(* PLC project Blank Project, Blank Blank 1.0 *)
(* stored: creationDateTime 2016-05-18T21:14:07, modificationDateTime 2020-07-06T15:08:10 *)

PROGRAM My_Program
  VAR
    flow_in AT %IW0 : INT;
    flow_out AT %IW1 : INT;
    ug_opcmd AT %QX0.0 : BOOL;
    ug_clcmd AT %QX0.1 : BOOL;
    ug_val AT %IW2 : INT;
    lg_opcmd AT %QX0.2 : BOOL;
    lg_clcmd AT %QX0.3 : BOOL;
    lg_val AT %IW3 : INT;
    uv_opcmd AT %QX0.4 : BOOL;
    uv_clcmd AT %QX0.5 : BOOL;
    uv_val AT %IW4 : INT;
    lv_opcmd AT %QX0.6 : BOOL;
    lv_clcmd AT %QX0.7 : BOOL;
    lv_val AT %IW5 : INT;
    dp_chmbr AT %IW6 : INT;
    dp_rsvr AT %IW7 : INT := 4200;
    dp_tlwtr AT %IW8 : INT;
    warn_btn AT %QX1.0 : BOOL;
    em_gt AT %QX1.1 : BOOL;
    em_vlv AT %QX1.2 : BOOL;
    ht_still AT %IW9 : INT := 2150;
    dprel_rsvr AT %QW0 : INT;
    rsrvr_eq AT %QX1.3 : BOOL;
    tlwtr_eq AT %QX1.4 : BOOL;
  END_VAR
  VAR
    TP0 : TP;
    TP1 : TP;
    TP2 : TP;
  END_VAR
  VAR  (* added by the conversion: wires and edge detectors of the diagram *)
    _XOR35_OUT : BOOL;
    _DIV140_OUT : REAL;
    _XOR28_OUT : BOOL;
    _DIV17_OUT : REAL;
    _XOR57_OUT : BOOL;
    _DIV144_OUT : REAL;
    _XOR83_OUT : BOOL;
    _DIV79_OUT : REAL;
  END_VAR

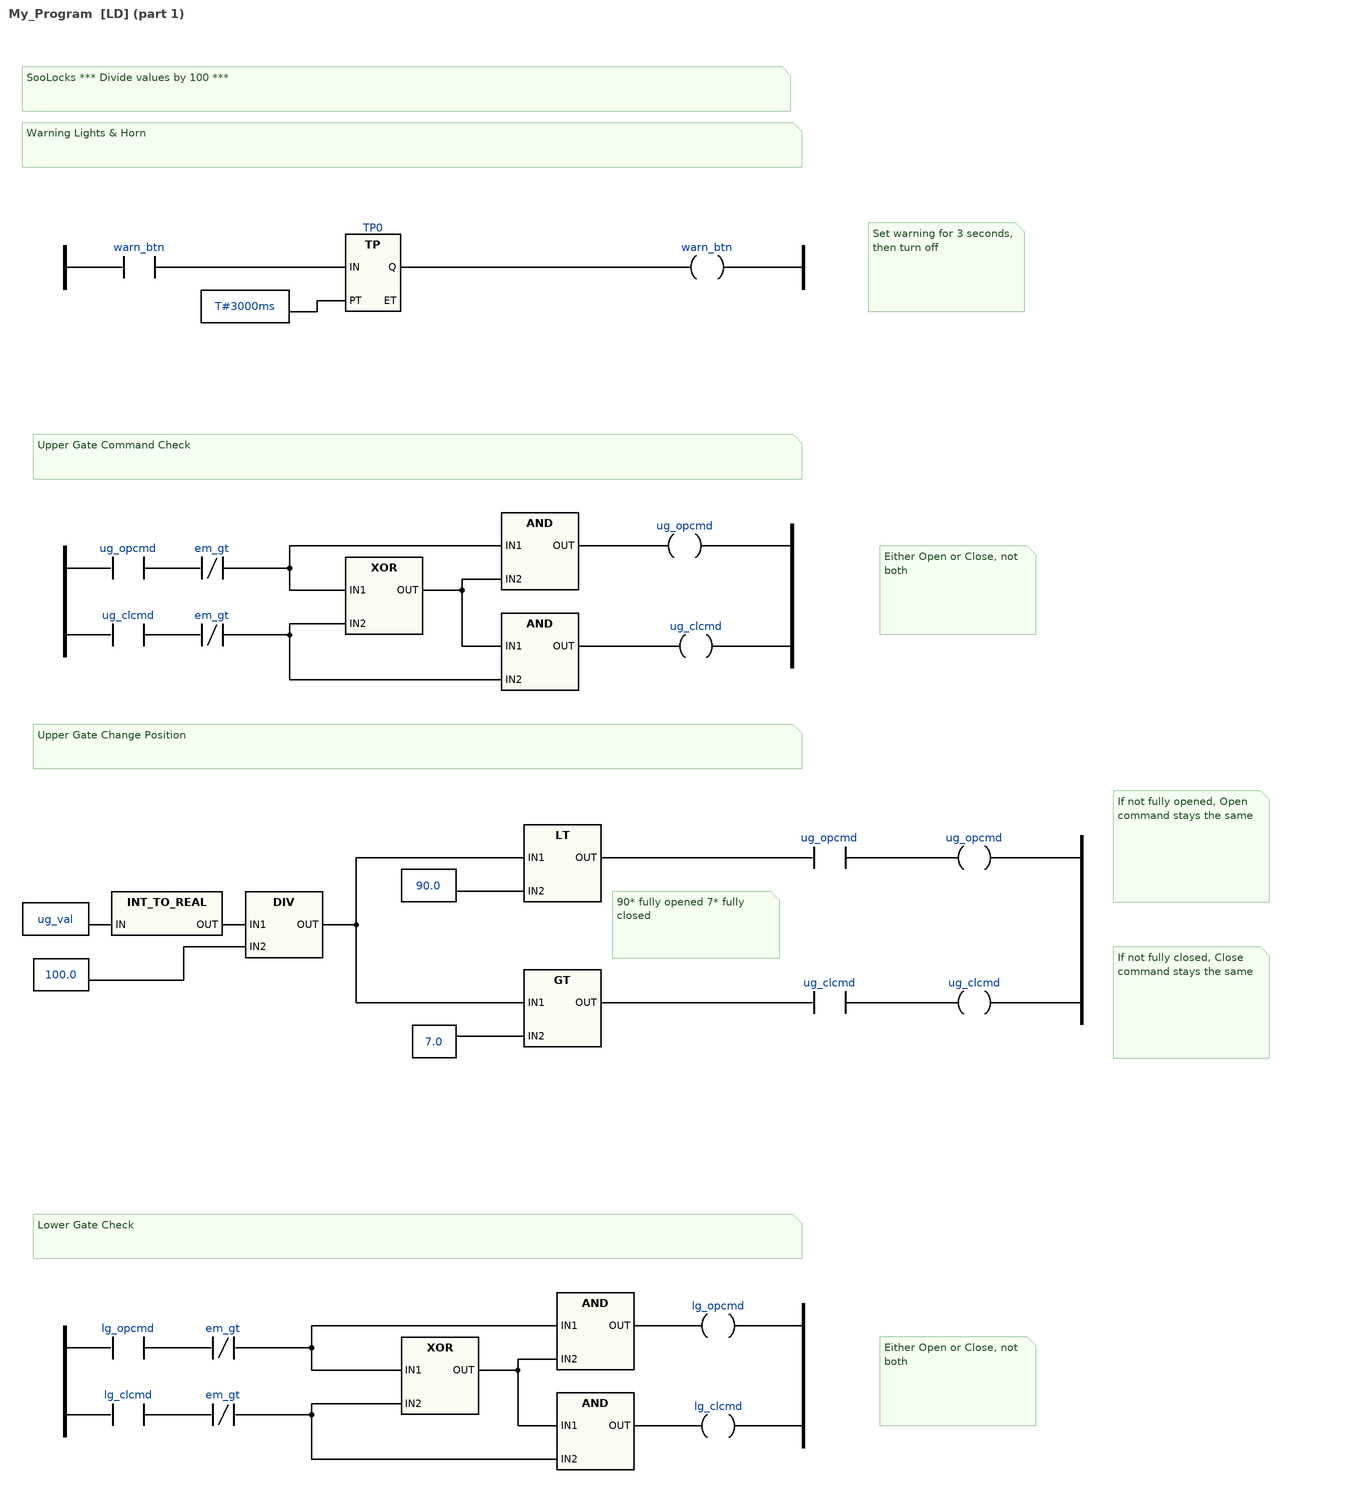
(* LD diagram, written out as Structured Text *)
(* SooLocks *** Divide values by 100 *** *)
(* Warning Lights & Horn *)
(* Set warning for 3 seconds, then turn off *)
TP0(IN := warn_btn, PT := T#3000ms);
warn_btn := TP0.Q;
(* Upper Gate Command Check *)
_XOR35_OUT := ug_opcmd AND NOT em_gt XOR ug_clcmd AND NOT em_gt;
ug_opcmd := ug_opcmd AND NOT em_gt AND _XOR35_OUT;
(* Either Open or Close, not both *)
ug_clcmd := _XOR35_OUT AND ug_clcmd AND NOT em_gt;
(* Upper Gate Change Position *)
(* If not fully opened, Open command stays the same *)
_DIV140_OUT := INT_TO_REAL(ug_val) / 100.0;
ug_opcmd := _DIV140_OUT < 90.0 AND ug_opcmd;
(* 90* fully opened 7* fully closed *)
(* If not fully closed, Close command stays the same *)
ug_clcmd := _DIV140_OUT > 7.0 AND ug_clcmd;
(* Lower Gate Check *)
_XOR28_OUT := lg_opcmd AND NOT em_gt XOR lg_clcmd AND NOT em_gt;
lg_opcmd := lg_opcmd AND NOT em_gt AND _XOR28_OUT;
(* Either Open or Close, not both *)
lg_clcmd := _XOR28_OUT AND lg_clcmd AND NOT em_gt;
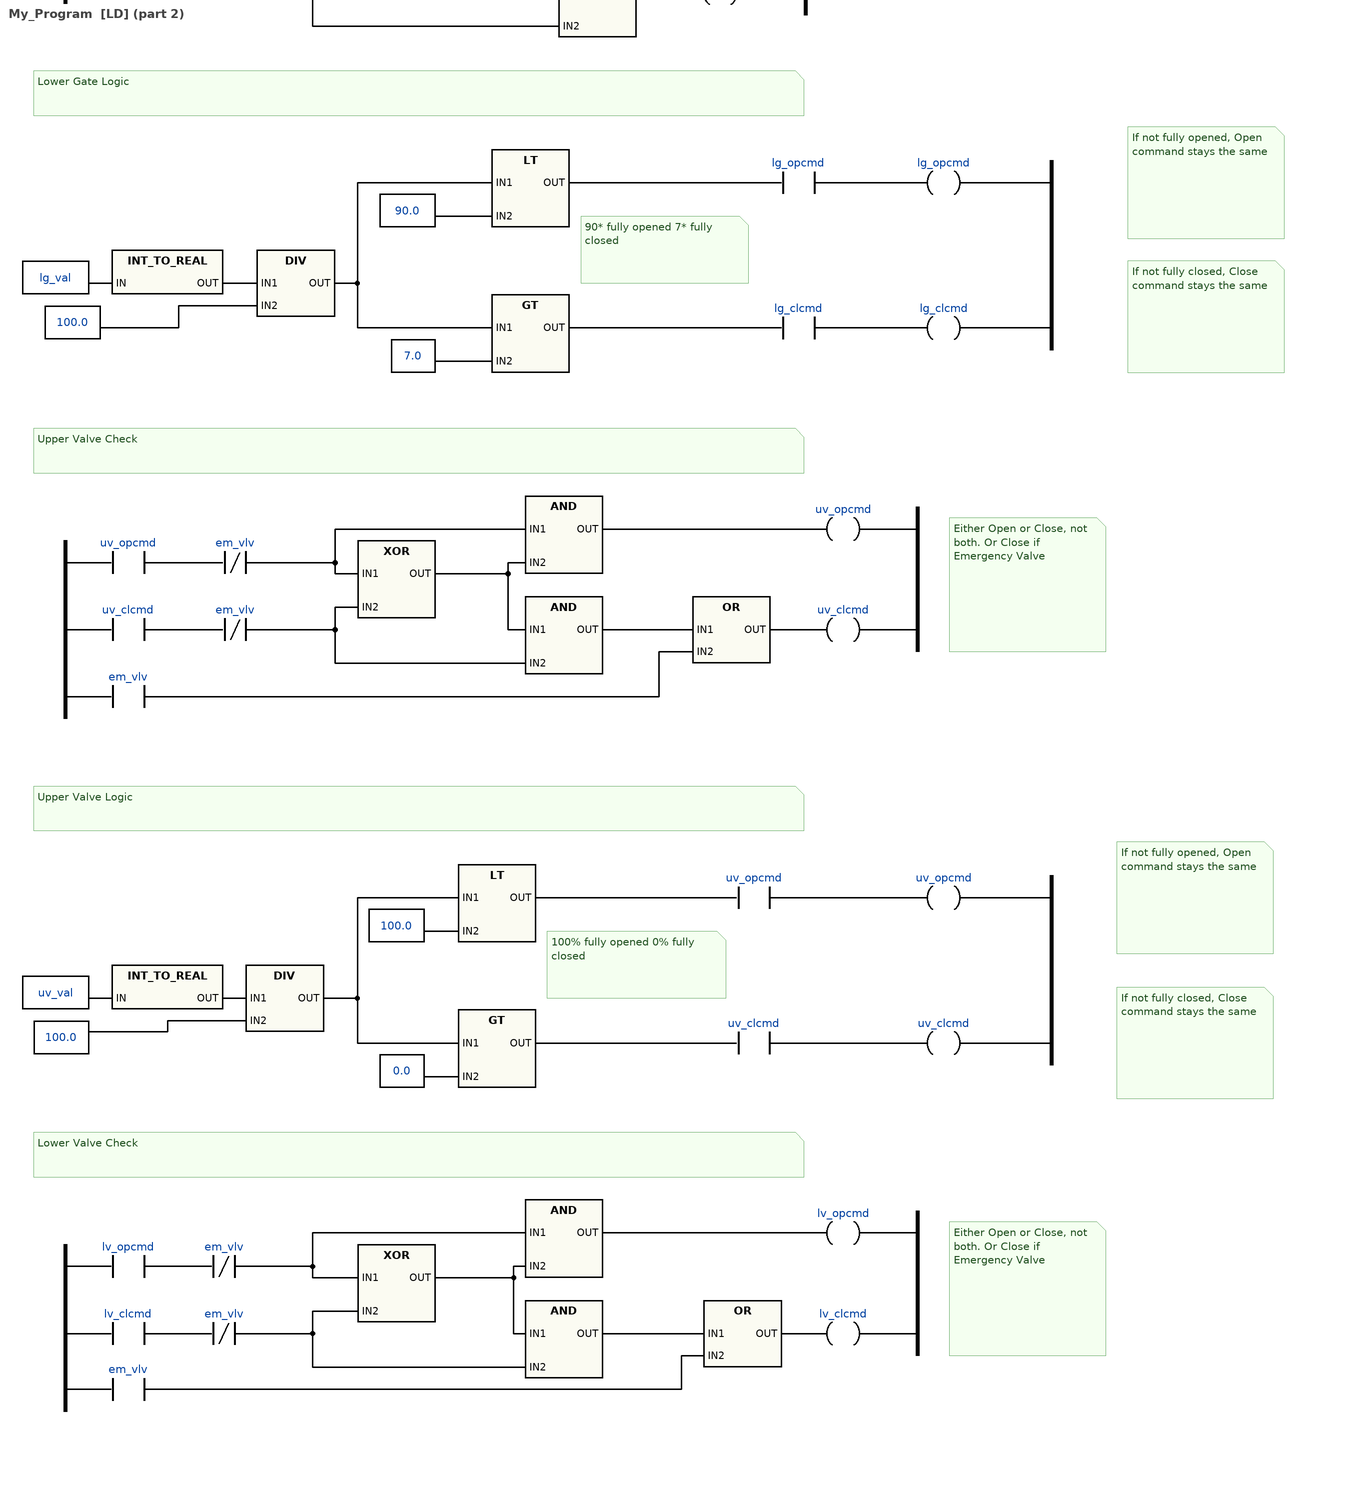
(* Lower Gate Logic *)
(* If not fully opened, Open command stays the same *)
_DIV17_OUT := INT_TO_REAL(lg_val) / 100.0;
lg_opcmd := _DIV17_OUT < 90.0 AND lg_opcmd;
(* 90* fully opened 7* fully closed *)
(* If not fully closed, Close command stays the same *)
lg_clcmd := _DIV17_OUT > 7.0 AND lg_clcmd;
(* Upper Valve Check *)
(* Either Open or Close, not both. Or Close if Emergency Valve *)
_XOR57_OUT := uv_opcmd AND NOT em_vlv XOR uv_clcmd AND NOT em_vlv;
uv_opcmd := uv_opcmd AND NOT em_vlv AND _XOR57_OUT;
uv_clcmd := _XOR57_OUT AND uv_clcmd AND NOT em_vlv OR em_vlv;
(* Upper Valve Logic *)
(* If not fully opened, Open command stays the same *)
_DIV144_OUT := INT_TO_REAL(uv_val) / 100.0;
uv_opcmd := _DIV144_OUT < 100.0 AND uv_opcmd;
(* 100% fully opened 0% fully closed *)
(* If not fully closed, Close command stays the same *)
uv_clcmd := _DIV144_OUT > 0.0 AND uv_clcmd;
(* Lower Valve Check *)
(* Either Open or Close, not both. Or Close if Emergency Valve *)
_XOR83_OUT := lv_opcmd AND NOT em_vlv XOR lv_clcmd AND NOT em_vlv;
lv_opcmd := lv_opcmd AND NOT em_vlv AND _XOR83_OUT;
lv_clcmd := _XOR83_OUT AND lv_clcmd AND NOT em_vlv OR em_vlv;
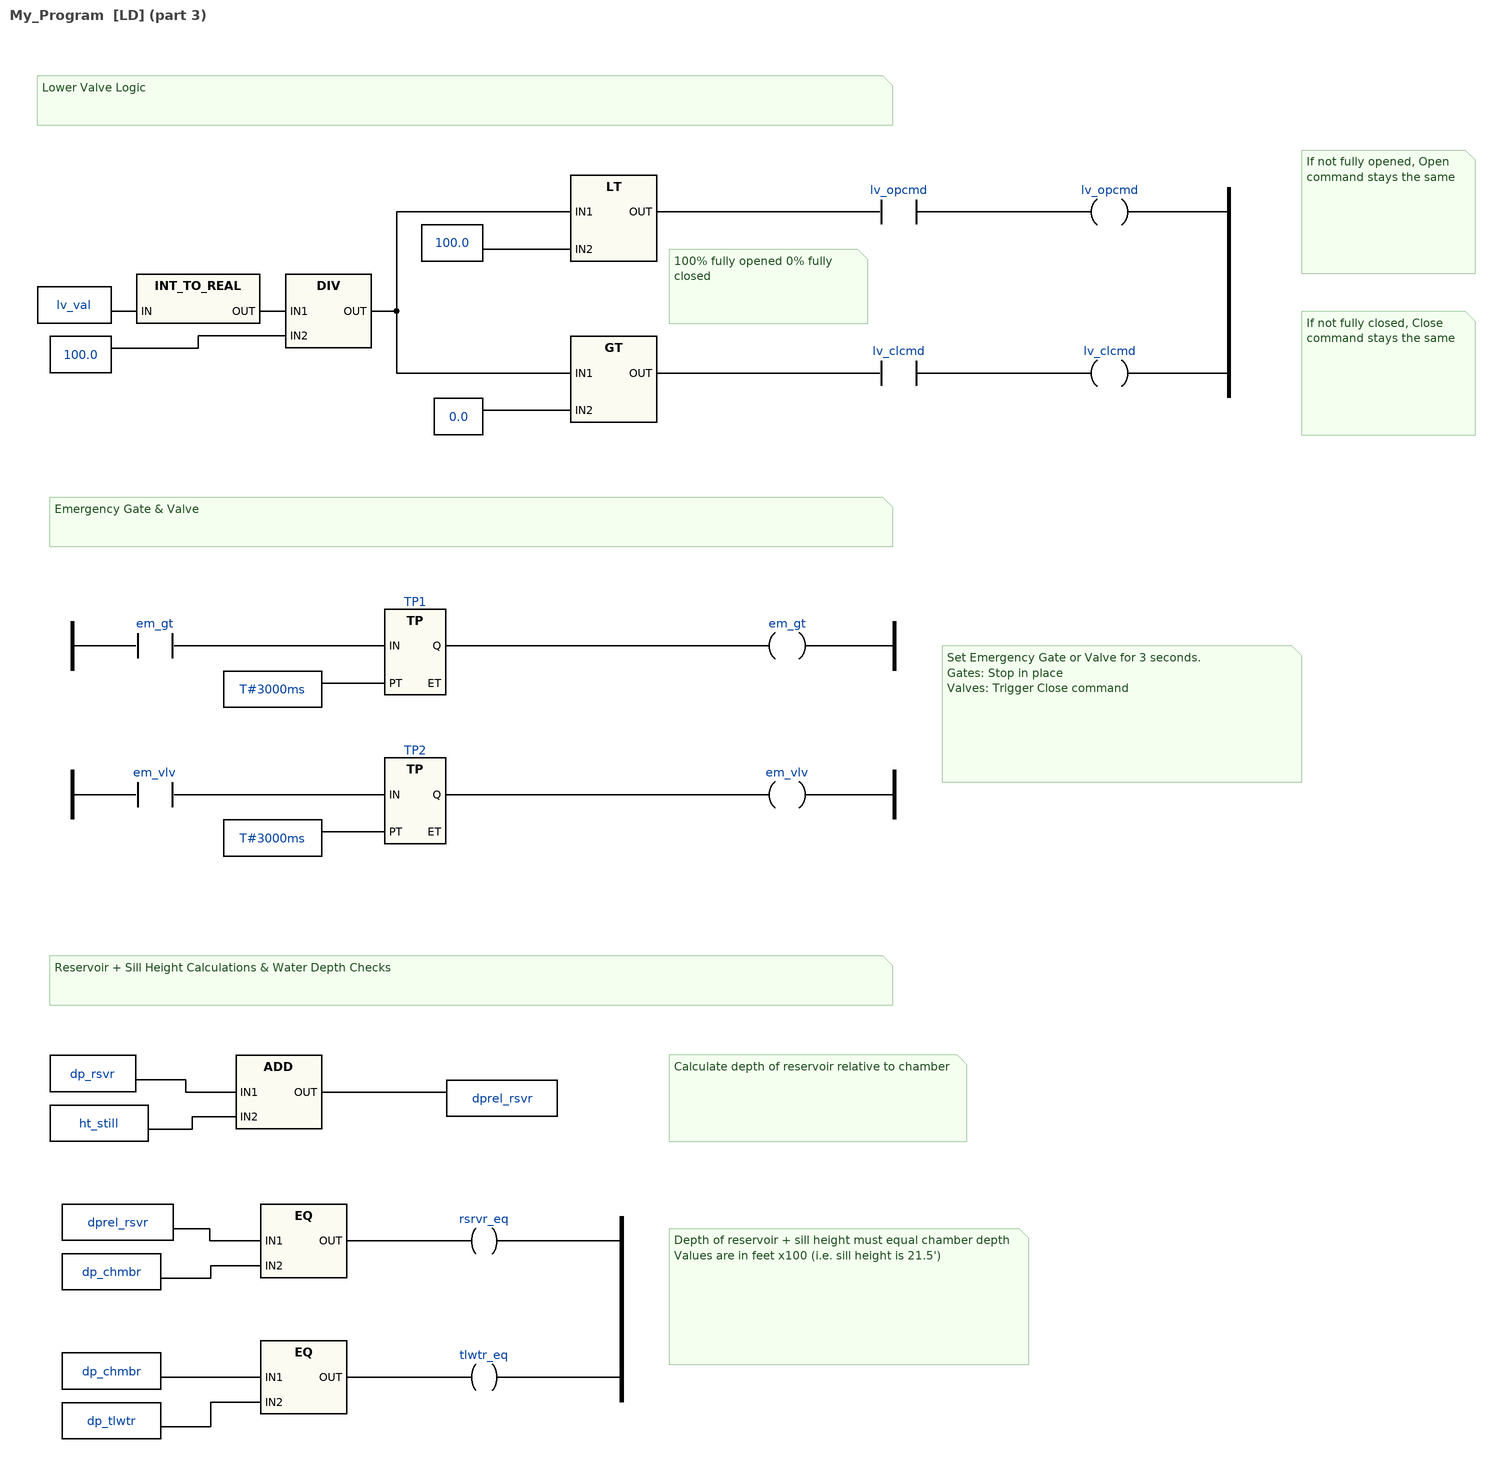
(* Lower Valve Logic *)
(* If not fully opened, Open command stays the same *)
_DIV79_OUT := INT_TO_REAL(lv_val) / 100.0;
lv_opcmd := _DIV79_OUT < 100.0 AND lv_opcmd;
(* 100% fully opened 0% fully closed *)
(* If not fully closed, Close command stays the same *)
lv_clcmd := _DIV79_OUT > 0.0 AND lv_clcmd;
(* Emergency Gate & Valve *)
TP1(IN := em_gt, PT := T#3000ms);
em_gt := TP1.Q;
(* Set Emergency Gate or Valve for 3 seconds. 
Gates: Stop in place
Valves: Trigger Close command *)
TP2(IN := em_vlv, PT := T#3000ms);
em_vlv := TP2.Q;
(* Reservoir + Sill Height Calculations & Water Depth Checks *)
(* Calculate depth of reservoir relative to chamber *)
dprel_rsvr := dp_rsvr + ht_still;
(* Depth of reservoir + sill height must equal chamber depth
Values are in feet x100 (i.e. sill height is 21.5') *)
rsrvr_eq := dprel_rsvr = dp_chmbr;
tlwtr_eq := dp_chmbr = dp_tlwtr;
END_PROGRAM

CONFIGURATION Config0
  RESOURCE Res0 ON PLC
    TASK TaskMain(INTERVAL := T#50ms, PRIORITY := 0);
    PROGRAM Inst0 WITH TaskMain : My_Program;
  END_RESOURCE
END_CONFIGURATION
